// TIA Portal V19 export
FUNCTION_BLOCK "FeedMachine_FB"   // FB25, LAD
TITLE = FEEDING AXIS MACHINE
// stored: Access Published, MemoryReserve 100, SetENOAutomatically false
   VAR_INPUT
      AreaInterface : "AreaInterface";
      ZSI : "udt_ZoneSafetyInterface";
      DSI : "udt_DeviceSafetyInterface";
      Drive : "TAx_DriveInterface";
      DataIn : "FeedMachine_DataIn";
      CIn : "FeedMachine_CIn";
      Config : "FeedMachine_Config";
   END_VAR
   VAR_OUTPUT
      MachineInterface : "MachineInterface";
      DataOut : "FeedMachine_DataOut";
      COut : "FeedMachine_COut";
   END_VAR
   VAR_IN_OUT
      TO_Ax : TO_SpeedAxis;
      Par : "FeedMachine_Par";
      Alarm : "FeedMachine_Alr";
      Warning : "FeedMachine_Wng";
   END_VAR
   VAR
      Sts : Struct
         Standstill : Bool := TRUE;
         AlarmPresence : Bool := FALSE;
         WarningPresence : Bool := FALSE;
         Gen_Cnd : Bool;
         Bwd_Cnd : Bool := FALSE;
         Fwd_Cnd : Bool := FALSE;
         ReductionRatio : LReal := 1.0;
      END_STRUCT;
      Ctrl : Struct
         StopDueDoorOpeningRequest : Bool;
         StopInPhase : Bool;
         StopProgrammed : Bool;
         StopAborting : Bool;
         Man_HighSpeed : Bool;
         Bwd_Man : Bool;
         Fwd_Man : Bool;
         Bwd_Aut : Bool;
         Fwd_Aut : Bool;
         Fan : Bool;
         Vel : LReal;
         Acc : LReal;
         Dec : LReal;
         Jerk : LReal;
      END_STRUCT;
      Diag : Struct
         Ax : "TO_Diagnostic";
      END_STRUCT;
      Ax : "SpeedAxis";
      Fan_M : "Motor";
      TON_NoPendingCmd : TON_TIME;
      TON_Feed_DelayManChangeSpeed : TON_TIME;
      TON_MissingCndBwd { S7_SetPoint := 'True'} : TON_TIME;
      TON_MissingCndFwd { S7_SetPoint := 'True'} : TON_TIME;
      TON_Fan_DelayOff : TON_TIME;
      TON_Brake_TimeOut { S7_SetPoint := 'True'} : TON_TIME;
      AUX : Struct
         PB_Bwd : Bool;
         PB_Fwd : Bool;
      END_STRUCT;
   END_VAR
   VAR_TEMP
      PE : Struct
         PB_Bwd : Bool;
         PB_Fwd : Bool;
      END_STRUCT;
      Req : Bool;
      AxisVelMax : LReal;
      LimVel_EngUnit : LReal;
      LimAcc_EngUnit : LReal;
      LimDec_EngUnit : LReal;
      LimJerk_EngUnit : LReal;
      Real_VelTarget : LReal;
   END_VAR
   VAR_TEMP   // added for the SCL form of the ladder/FBD networks
      _w1 : Bool;
      _w2 : Bool;
   END_VAR
BEGIN

REGION Network 1 (SCL): Reset
   IF #AreaInterface.RstAlarms THEN

       #Alarm.BrakeTimeOut :=

       #Warning.NotAutReady :=
       #Warning.MissingCnd_Bkw :=
       #Warning.MissingCnd_Fwd := FALSE;
   END_IF;
END_REGION

REGION Network 2: Alarm motor brake timeout
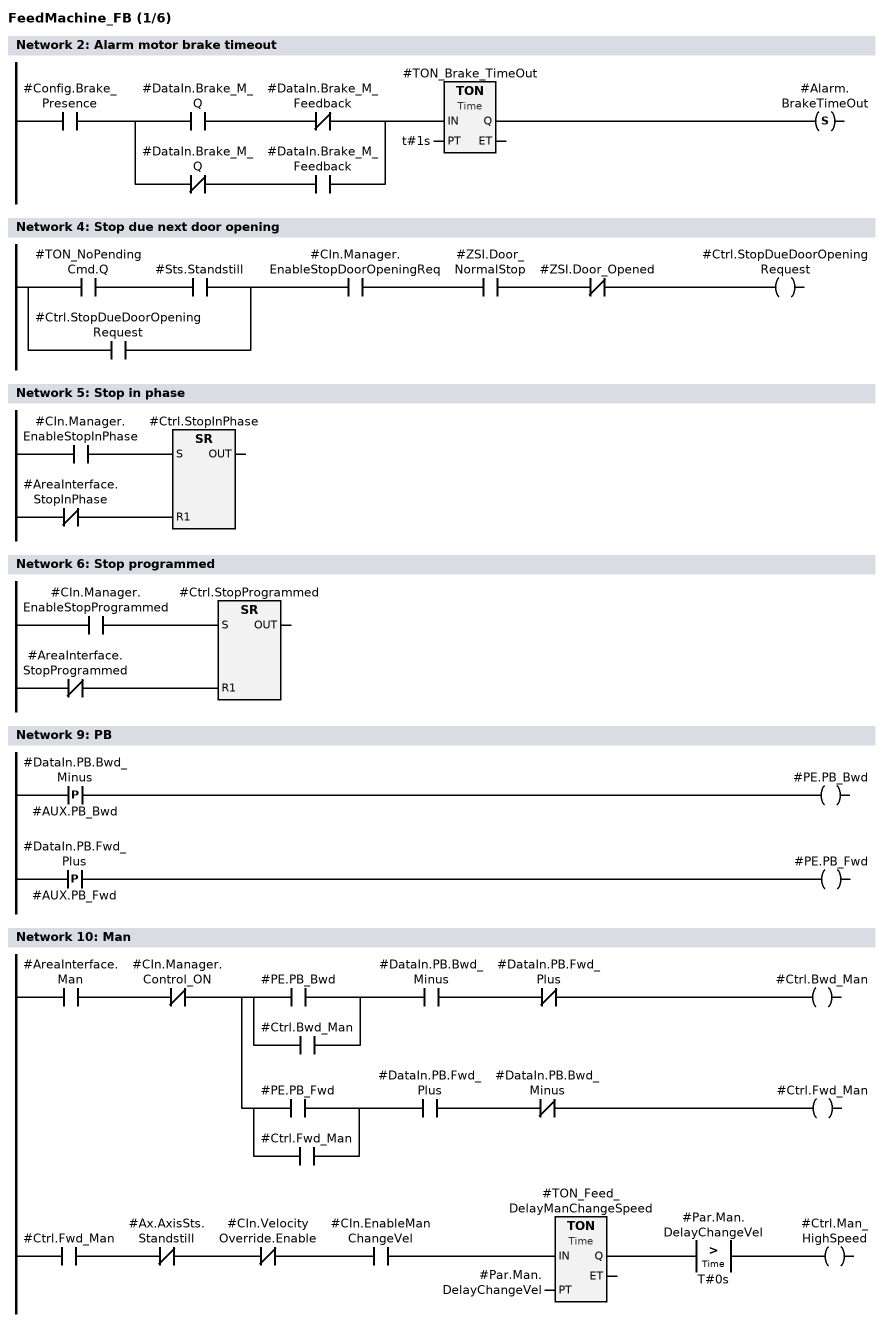
   RUNG wire#powerrail
      Contact( #Config.Brake_Presence )
      wire#w1
      Contact( #DataIn.Brake_M_Q )
      I_Contact( #DataIn.Brake_M_Feedback )
      wire#w2
      { S7_Templates := "time_type := Time" } #TON_Brake_TimeOut.TON(pt := t#1s, et =>)
      S_Coil( #Alarm.BrakeTimeOut )
   END_RUNG
   RUNG wire#w1
      I_Contact( #DataIn.Brake_M_Q )
      Contact( #DataIn.Brake_M_Feedback )
   END_RUNG wire#w2
   // the same network as SCL:
   #TON_Brake_TimeOut(IN := #Config.Brake_Presence AND ((#DataIn.Brake_M_Q AND NOT #DataIn.Brake_M_Feedback) OR (NOT #DataIn.Brake_M_Q AND #DataIn.Brake_M_Feedback)),   // TON
                      PT := t#1s);
   IF #TON_Brake_TimeOut.Q THEN #Alarm.BrakeTimeOut := TRUE; END_IF;
END_REGION

REGION Network 3: <<< MACHINE STOP >>>
END_REGION

REGION Network 4: Stop due next door opening
   RUNG wire#powerrail
      Contact( #TON_NoPendingCmd.Q )
      Contact( #Sts.Standstill )
      wire#w1
      Contact( #CIn.Manager.EnableStopDoorOpeningReq )
      Contact( #ZSI.Door_NormalStop )
      I_Contact( #ZSI.Door_Opened )
      Coil( #Ctrl.StopDueDoorOpeningRequest )
   END_RUNG
   RUNG wire#powerrail
      Contact( #Ctrl.StopDueDoorOpeningRequest )
   END_RUNG wire#w1
   // the same network as SCL:
   #Ctrl.StopDueDoorOpeningRequest := ((#TON_NoPendingCmd.Q AND #Sts.Standstill) OR #Ctrl.StopDueDoorOpeningRequest) AND #CIn.Manager.EnableStopDoorOpeningReq AND #ZSI.Door_NormalStop AND NOT #ZSI.Door_Opened;
END_REGION

REGION Network 5: Stop in phase
   RUNG wire#powerrail
      Contact( #CIn.Manager.EnableStopInPhase )
      S_SR(operand := #Ctrl.StopInPhase, r1 := wire#w1)
   END_RUNG
   RUNG wire#powerrail
      I_Contact( #AreaInterface.StopInPhase )
   END_RUNG wire#w1
   // the same network as SCL:
   IF #CIn.Manager.EnableStopInPhase THEN
       #Ctrl.StopInPhase := TRUE;   // SR flip-flop
   END_IF;
   IF NOT #AreaInterface.StopInPhase THEN #Ctrl.StopInPhase := FALSE; END_IF;
END_REGION

REGION Network 6: Stop programmed
   RUNG wire#powerrail
      Contact( #CIn.Manager.EnableStopProgrammed )
      S_SR(operand := #Ctrl.StopProgrammed, r1 := wire#w1)
   END_RUNG
   RUNG wire#powerrail
      I_Contact( #AreaInterface.StopProgrammed )
   END_RUNG wire#w1
   // the same network as SCL:
   IF #CIn.Manager.EnableStopProgrammed THEN
       #Ctrl.StopProgrammed := TRUE;   // SR flip-flop
   END_IF;
   IF NOT #AreaInterface.StopProgrammed THEN #Ctrl.StopProgrammed := FALSE; END_IF;
END_REGION

REGION Network 7: >
END_REGION

REGION Network 8: <<< FEED >>>
END_REGION

REGION Network 9: PB
   RUNG wire#powerrail
      P_Contact(operand := #DataIn.PB.Bwd_Minus, bit := #AUX.PB_Bwd)
      Coil( #PE.PB_Bwd )
   END_RUNG
   RUNG wire#powerrail
      P_Contact(operand := #DataIn.PB.Fwd_Plus, bit := #AUX.PB_Fwd)
      Coil( #PE.PB_Fwd )
   END_RUNG
   // the same network as SCL:
   #_w1 := #DataIn.PB.Bwd_Minus AND NOT #AUX.PB_Bwd;   // rising edge of #DataIn.PB.Bwd_Minus
   #AUX.PB_Bwd := #DataIn.PB.Bwd_Minus;
   #PE.PB_Bwd := #_w1;
   #_w2 := #DataIn.PB.Fwd_Plus AND NOT #AUX.PB_Fwd;   // rising edge of #DataIn.PB.Fwd_Plus
   #AUX.PB_Fwd := #DataIn.PB.Fwd_Plus;
   #PE.PB_Fwd := #_w2;
END_REGION

REGION Network 10: Man
   RUNG wire#powerrail
      Contact( #AreaInterface.Man )
      I_Contact( #CIn.Manager.Control_ON )
      wire#w1
      Contact( #PE.PB_Bwd )
      wire#w2
      Contact( #DataIn.PB.Bwd_Minus )
      I_Contact( #DataIn.PB.Fwd_Plus )
      Coil( #Ctrl.Bwd_Man )
   END_RUNG
   RUNG wire#w1
      Contact( #Ctrl.Bwd_Man )
   END_RUNG wire#w2
   RUNG wire#w1
      Contact( #PE.PB_Fwd )
      wire#w3
      Contact( #DataIn.PB.Fwd_Plus )
      I_Contact( #DataIn.PB.Bwd_Minus )
      Coil( #Ctrl.Fwd_Man )
   END_RUNG
   RUNG wire#w1
      Contact( #Ctrl.Fwd_Man )
   END_RUNG wire#w3
   RUNG wire#powerrail
      Contact( #Ctrl.Fwd_Man )
      I_Contact( #Ax.AxisSts.Standstill )
      I_Contact( #CIn.VelocityOverride.Enable )
      Contact( #CIn.EnableManChangeVel )
      { S7_Templates := "time_type := Time" } #TON_Feed_DelayManChangeSpeed.TON(pt := #Par.Man.DelayChangeVel, et =>)
      { S7_Templates := "SrcType := Time" } GT_Contact(in1 := #Par.Man.DelayChangeVel, in2 := T#0s)
      Coil( #Ctrl.Man_HighSpeed )
   END_RUNG
   // the same network as SCL:
   #_w1 := #AreaInterface.Man AND NOT #CIn.Manager.Control_ON;
   #Ctrl.Bwd_Man := #_w1 AND (#PE.PB_Bwd OR #Ctrl.Bwd_Man) AND #DataIn.PB.Bwd_Minus AND NOT #DataIn.PB.Fwd_Plus;
   #Ctrl.Fwd_Man := #_w1 AND (#PE.PB_Fwd OR #Ctrl.Fwd_Man) AND #DataIn.PB.Fwd_Plus AND NOT #DataIn.PB.Bwd_Minus;
   #TON_Feed_DelayManChangeSpeed(IN := #Ctrl.Fwd_Man AND NOT #Ax.AxisSts.Standstill AND NOT #CIn.VelocityOverride.Enable AND #CIn.EnableManChangeVel,   // TON
                           PT := #Par.Man.DelayChangeVel);
   #Ctrl.Man_HighSpeed := #TON_Feed_DelayManChangeSpeed.Q AND (#Par.Man.DelayChangeVel > T#0s);
END_REGION

REGION Network 11: Aut
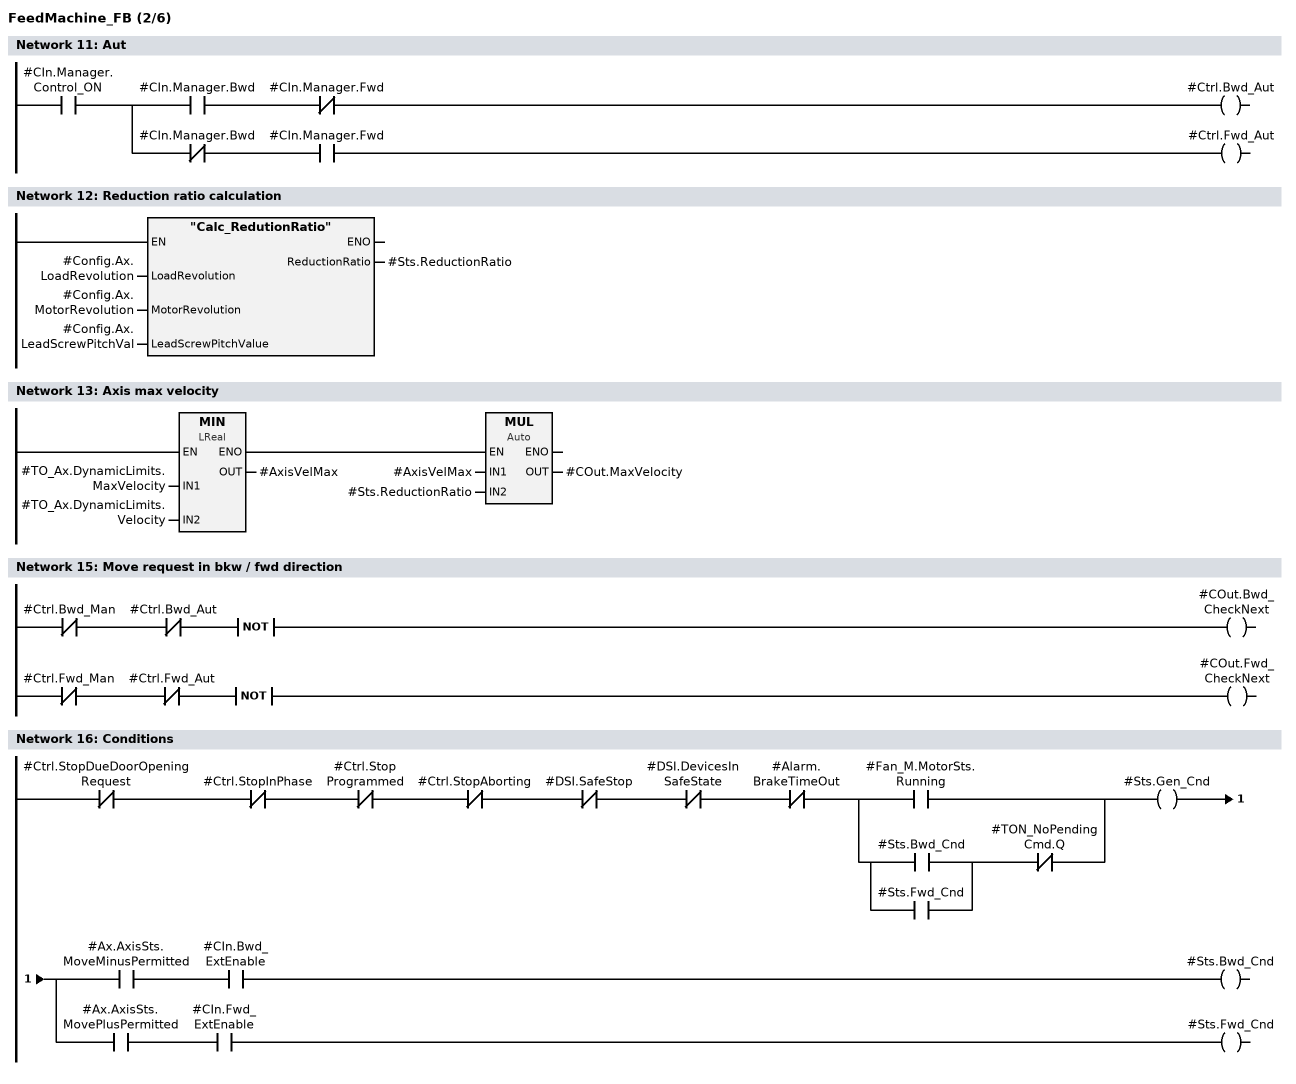
   RUNG wire#powerrail
      Contact( #CIn.Manager.Control_ON )
      wire#w1
      Contact( #CIn.Manager.Bwd )
      I_Contact( #CIn.Manager.Fwd )
      Coil( #Ctrl.Bwd_Aut )
   END_RUNG
   RUNG wire#w1
      I_Contact( #CIn.Manager.Bwd )
      Contact( #CIn.Manager.Fwd )
      Coil( #Ctrl.Fwd_Aut )
   END_RUNG
   // the same network as SCL:
   #Ctrl.Bwd_Aut := #CIn.Manager.Control_ON AND #CIn.Manager.Bwd AND NOT #CIn.Manager.Fwd;
   #Ctrl.Fwd_Aut := #CIn.Manager.Control_ON AND NOT #CIn.Manager.Bwd AND #CIn.Manager.Fwd;
END_REGION

REGION Network 12: Reduction ratio calculation
   RUNG wire#powerrail
      "Calc_RedutionRatio"(LoadRevolution := #Config.Ax.LoadRevolution, MotorRevolution := #Config.Ax.MotorRevolution, LeadScrewPitchValue := #Config.Ax.LeadScrewPitchVal, ReductionRatio => #Sts.ReductionRatio)
   END_RUNG
   // the same network as SCL:
   "Calc_RedutionRatio"(LoadRevolution := #Config.Ax.LoadRevolution,
                        MotorRevolution := #Config.Ax.MotorRevolution,
                        LeadScrewPitchValue := #Config.Ax.LeadScrewPitchVal,
                        ReductionRatio => #Sts.ReductionRatio);
END_REGION

REGION Network 13: Axis max velocity
   RUNG wire#powerrail
      { S7_Templates := "[card := 2, value_type := LReal]" } MIN(in1 := #TO_Ax.DynamicLimits.MaxVelocity, in2 := #TO_Ax.DynamicLimits.Velocity, out => #AxisVelMax)
      Mul(in1 := #AxisVelMax, in2 := #Sts.ReductionRatio, out => #COut.MaxVelocity)
   END_RUNG
   // the same network as SCL:
   #AxisVelMax := MIN(IN1 := #TO_Ax.DynamicLimits.MaxVelocity, IN2 := #TO_Ax.DynamicLimits.Velocity);
   #COut.MaxVelocity := #AxisVelMax * #Sts.ReductionRatio;
END_REGION

REGION Network 14 (SCL): Velocity & Dynamics
   #LimVel_EngUnit := #TO_Ax.DynamicLimits.MaxVelocity *  #Sts.ReductionRatio;
   #LimAcc_EngUnit := #TO_Ax.DynamicLimits.MaxAcceleration * #Sts.ReductionRatio;
   #LimDec_EngUnit := #TO_Ax.DynamicLimits.MaxDeceleration * #Sts.ReductionRatio;
   #LimJerk_EngUnit := #TO_Ax.DynamicLimits.MaxJerk * #Sts.ReductionRatio;




   #Ctrl.Vel := 0.0;

   IF #Ctrl.Bwd_Man AND #Ax.AxisCtrl.MoveMinus THEN


       #Ctrl.Acc := #Par.Man.Acc;
       #Ctrl.Dec := #Par.Man.Dec;
       #Ctrl.Jerk := #Par.Man.Jerk;

       #Ctrl.Vel := #Par.Man.VelBwd;

   ELSIF #Ctrl.Fwd_Man AND #Ax.AxisCtrl.MovePlus THEN


       #Ctrl.Acc := #Par.Man.Acc;
       #Ctrl.Dec := #Par.Man.Dec;
       #Ctrl.Jerk := #Par.Man.Jerk;


       IF #Ctrl.Man_HighSpeed THEN
           #Ctrl.Vel := #Par.Man.VelFwdHigh;
       ELSE
           #Ctrl.Vel := #Par.Man.VelFwdLow;
       END_IF;


   ELSIF (#Ctrl.Bwd_Aut AND #Ax.AxisCtrl.MoveMinus) OR (#Ctrl.Fwd_Aut AND #Ax.AxisCtrl.MovePlus)  THEN

       #Ctrl.Vel := #CIn.Manager.Vel;
       #Ctrl.Acc := #CIn.Manager.Acc;
       #Ctrl.Dec := #CIn.Manager.Dec;
       #Ctrl.Jerk := #CIn.Manager.Jerk;

   END_IF;


   // Dynamics limit

   #Ctrl.Vel := MIN(IN1:= #Ctrl.Vel,IN2:= #LimVel_EngUnit);

   #Ctrl.Acc := MIN(IN1:= #Ctrl.Acc,IN2:= #LimAcc_EngUnit);
   IF #Ctrl.Acc <= 0.0 THEN
       #Ctrl.Acc := #Par.Man.Acc;
   END_IF;

   #Ctrl.Dec := MIN(IN1:= #Ctrl.Dec,IN2:= #LimDec_EngUnit);
   IF #Ctrl.Dec <= 0.0 THEN
       #Ctrl.Dec := #Par.Man.Dec;
   END_IF;

   IF #Ctrl.Jerk > 0.0 THEN
       #Ctrl.Jerk := MIN(IN1:= #Ctrl.Jerk,IN2:= #LimJerk_EngUnit);
   ELSE
       #Ctrl.Jerk := 0.0;
   END_IF;



   // Velocity override
   // 
   #TO_Ax.Override.Velocity := 100.0;
   IF #CIn.VelocityOverride.Enable THEN
       #TO_Ax.Override.Velocity := LIMIT(MN:= 1.0, IN:=#CIn.VelocityOverride.Value, MX:=100.0);
   END_IF;



   // SLS velocity limit
   //
   IF #ZSI.Door_Opened AND #Ctrl.Vel > #Config.SLS_VEL THEN
       #Ctrl.Vel := #Config.SLS_VEL;
   END_IF;



   // Conversion and write dynamics value
   // 
   #Ax.AxisCtrl.Velocity := #Ctrl.Vel / #Sts.ReductionRatio;
   #Ax.AxisCtrl.Acceleration := #Ctrl.Acc / #Sts.ReductionRatio;
   #Ax.AxisCtrl.Deceleration := #Ctrl.Dec / #Sts.ReductionRatio;
   #Ax.AxisCtrl.Jerk := #Ctrl.Jerk / #Sts.ReductionRatio;

   #Ax.StandtillVelocity := #Config.Ax.StandstillVelocity / #Sts.ReductionRatio;
END_REGION

REGION Network 15: Move request in bkw / fwd direction
   RUNG wire#powerrail
      I_Contact( #Ctrl.Bwd_Man )
      I_Contact( #Ctrl.Bwd_Aut )
      Not()
      Coil( #COut.Bwd_CheckNext )
   END_RUNG
   RUNG wire#powerrail
      I_Contact( #Ctrl.Fwd_Man )
      I_Contact( #Ctrl.Fwd_Aut )
      Not()
      Coil( #COut.Fwd_CheckNext )
   END_RUNG
   // the same network as SCL:
   #COut.Bwd_CheckNext := NOT (NOT #Ctrl.Bwd_Man AND NOT #Ctrl.Bwd_Aut);
   #COut.Fwd_CheckNext := NOT (NOT #Ctrl.Fwd_Man AND NOT #Ctrl.Fwd_Aut);
END_REGION

REGION Network 16: Conditions
   RUNG wire#powerrail
      I_Contact( #Ctrl.StopDueDoorOpeningRequest )
      I_Contact( #Ctrl.StopInPhase )
      I_Contact( #Ctrl.StopProgrammed )
      I_Contact( #Ctrl.StopAborting )
      I_Contact( #DSI.SafeStop )
      I_Contact( #DSI.DevicesInSafeState )
      I_Contact( #Alarm.BrakeTimeOut )
      wire#w1
      Contact( #Fan_M.MotorSts.Running )
      wire#w2
      Coil( #Sts.Gen_Cnd )
      wire#w4
      Contact( #Ax.AxisSts.MoveMinusPermitted )
      Contact( #CIn.Bwd_ExtEnable )
      Coil( #Sts.Bwd_Cnd )
   END_RUNG
   RUNG wire#w1
      Contact( #Sts.Bwd_Cnd )
      wire#w3
      I_Contact( #TON_NoPendingCmd.Q )
   END_RUNG wire#w2
   RUNG wire#w1
      Contact( #Sts.Fwd_Cnd )
   END_RUNG wire#w3
   RUNG wire#w4
      Contact( #Ax.AxisSts.MovePlusPermitted )
      Contact( #CIn.Fwd_ExtEnable )
      Coil( #Sts.Fwd_Cnd )
   END_RUNG
   // the same network as SCL:
   #Sts.Gen_Cnd := NOT #Ctrl.StopDueDoorOpeningRequest AND NOT #Ctrl.StopInPhase AND NOT #Ctrl.StopProgrammed AND NOT #Ctrl.StopAborting AND NOT #DSI.SafeStop AND NOT #DSI.DevicesInSafeState AND NOT #Alarm.BrakeTimeOut AND (#Fan_M.MotorSts.Running OR ((#Sts.Bwd_Cnd OR #Sts.Fwd_Cnd) AND NOT #TON_NoPendingCmd.Q));
   #Sts.Bwd_Cnd := #Sts.Gen_Cnd AND #Ax.AxisSts.MoveMinusPermitted AND #CIn.Bwd_ExtEnable;
   #Sts.Fwd_Cnd := #Sts.Gen_Cnd AND #Ax.AxisSts.MovePlusPermitted AND #CIn.Fwd_ExtEnable;
END_REGION

REGION Network 17: Missing conditions
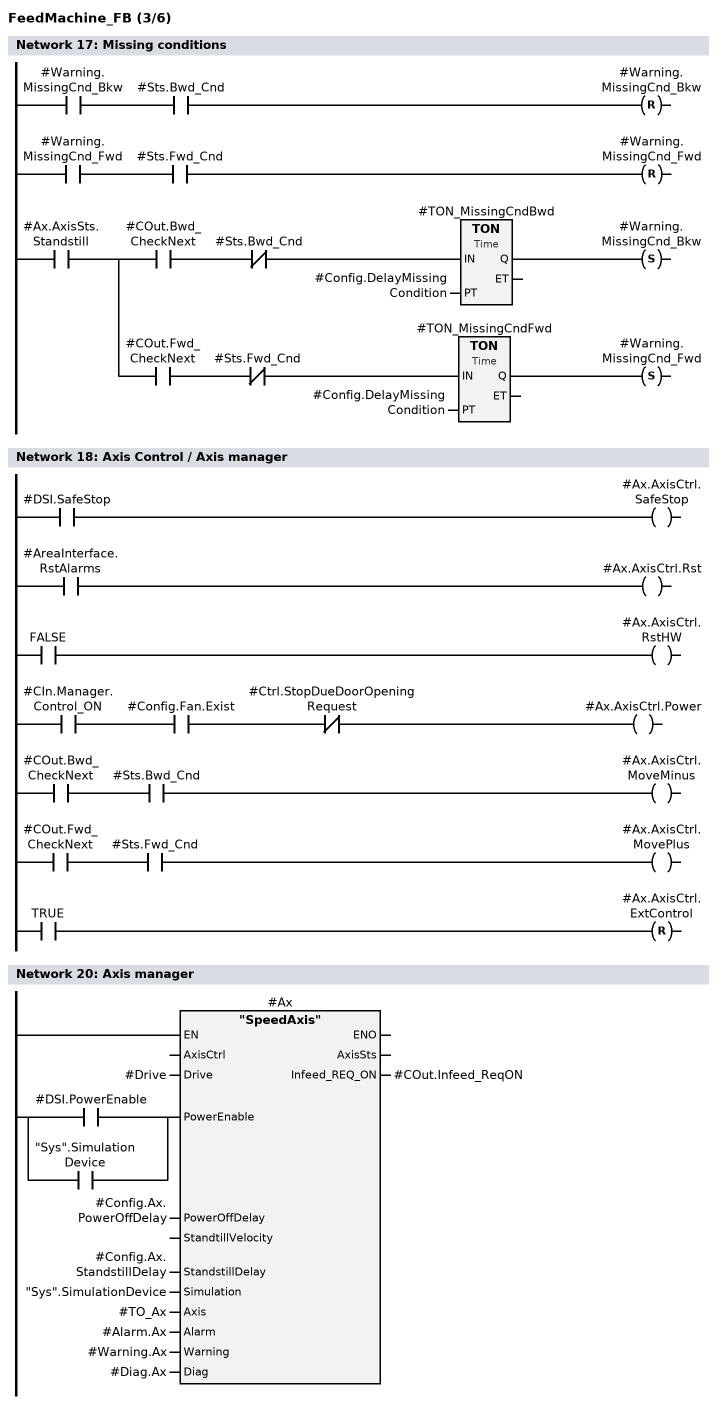
   RUNG wire#powerrail
      Contact( #Warning.MissingCnd_Bkw )
      Contact( #Sts.Bwd_Cnd )
      R_Coil( #Warning.MissingCnd_Bkw )
   END_RUNG
   RUNG wire#powerrail
      Contact( #Warning.MissingCnd_Fwd )
      Contact( #Sts.Fwd_Cnd )
      R_Coil( #Warning.MissingCnd_Fwd )
   END_RUNG
   RUNG wire#powerrail
      Contact( #Ax.AxisSts.Standstill )
      wire#w1
      Contact( #COut.Bwd_CheckNext )
      I_Contact( #Sts.Bwd_Cnd )
      { S7_Templates := "time_type := Time" } #TON_MissingCndBwd.TON(pt := #Config.DelayMissingCondition, et =>)
      S_Coil( #Warning.MissingCnd_Bkw )
   END_RUNG
   RUNG wire#w1
      Contact( #COut.Fwd_CheckNext )
      I_Contact( #Sts.Fwd_Cnd )
      { S7_Templates := "time_type := Time" } #TON_MissingCndFwd.TON(pt := #Config.DelayMissingCondition, et =>)
      S_Coil( #Warning.MissingCnd_Fwd )
   END_RUNG
   // the same network as SCL:
   IF #Warning.MissingCnd_Bkw AND #Sts.Bwd_Cnd THEN #Warning.MissingCnd_Bkw := FALSE; END_IF;
   IF #Warning.MissingCnd_Fwd AND #Sts.Fwd_Cnd THEN #Warning.MissingCnd_Fwd := FALSE; END_IF;
   #TON_MissingCndBwd(IN := #Ax.AxisSts.Standstill AND #COut.Bwd_CheckNext AND NOT #Sts.Bwd_Cnd,   // TON
                      PT := #Config.DelayMissingCondition);
   IF #TON_MissingCndBwd.Q THEN #Warning.MissingCnd_Bkw := TRUE; END_IF;
   #TON_MissingCndFwd(IN := #Ax.AxisSts.Standstill AND #COut.Fwd_CheckNext AND NOT #Sts.Fwd_Cnd,   // TON
                      PT := #Config.DelayMissingCondition);
   IF #TON_MissingCndFwd.Q THEN #Warning.MissingCnd_Fwd := TRUE; END_IF;
END_REGION

REGION Network 18: Axis Control / Axis manager
   RUNG wire#powerrail
      Contact( #DSI.SafeStop )
      Coil( #Ax.AxisCtrl.SafeStop )
   END_RUNG
   RUNG wire#powerrail
      Contact( #AreaInterface.RstAlarms )
      Coil( #Ax.AxisCtrl.Rst )
   END_RUNG
   RUNG wire#powerrail
      Contact( FALSE )
      Coil( #Ax.AxisCtrl.RstHW )
   END_RUNG
   RUNG wire#powerrail
      Contact( #CIn.Manager.Control_ON )
      Contact( #Config.Fan.Exist )
      I_Contact( #Ctrl.StopDueDoorOpeningRequest )
      Coil( #Ax.AxisCtrl.Power )
   END_RUNG
   RUNG wire#powerrail
      Contact( #COut.Bwd_CheckNext )
      Contact( #Sts.Bwd_Cnd )
      Coil( #Ax.AxisCtrl.MoveMinus )
   END_RUNG
   RUNG wire#powerrail
      Contact( #COut.Fwd_CheckNext )
      Contact( #Sts.Fwd_Cnd )
      Coil( #Ax.AxisCtrl.MovePlus )
   END_RUNG
   RUNG wire#powerrail
      Contact( TRUE )
      R_Coil( #Ax.AxisCtrl.ExtControl )
   END_RUNG
   // the same network as SCL:
   #Ax.AxisCtrl.SafeStop := #DSI.SafeStop;
   #Ax.AxisCtrl.Rst := #AreaInterface.RstAlarms;
   #Ax.AxisCtrl.RstHW := FALSE;
   #Ax.AxisCtrl.Power := #CIn.Manager.Control_ON AND #Config.Fan.Exist AND NOT #Ctrl.StopDueDoorOpeningRequest;
   #Ax.AxisCtrl.MoveMinus := #COut.Bwd_CheckNext AND #Sts.Bwd_Cnd;
   #Ax.AxisCtrl.MovePlus := #COut.Fwd_CheckNext AND #Sts.Fwd_Cnd;
   IF TRUE THEN #Ax.AxisCtrl.ExtControl := FALSE; END_IF;
END_REGION

REGION Network 20: Axis manager
   RUNG wire#powerrail
      #Ax(PowerEnable := wire#w1, AxisCtrl :=, Drive := #Drive, PowerOffDelay := #Config.Ax.PowerOffDelay, StandtillVelocity :=, StandstillDelay := #Config.Ax.StandstillDelay, Simulation := "Sys".SimulationDevice, Axis := #TO_Ax, Alarm := #Alarm.Ax, Warning := #Warning.Ax, Diag := #Diag.Ax, AxisSts =>, Infeed_REQ_ON => #COut.Infeed_ReqON)
   END_RUNG
   RUNG wire#powerrail
      Contact( #DSI.PowerEnable )
   END_RUNG wire#w1
   RUNG wire#powerrail
      Contact( "Sys".SimulationDevice )
   END_RUNG wire#w1
   // the same network as SCL:
   #Ax(Drive := #Drive,   // "SpeedAxis"
       PowerEnable := #DSI.PowerEnable OR "Sys".SimulationDevice,
       PowerOffDelay := #Config.Ax.PowerOffDelay,
       StandstillDelay := #Config.Ax.StandstillDelay,
       Simulation := "Sys".SimulationDevice,
       Axis := #TO_Ax,
       Alarm := #Alarm.Ax,
       Warning := #Warning.Ax,
       Diag := #Diag.Ax,
       Infeed_REQ_ON => #COut.Infeed_ReqON);
END_REGION

REGION Network 21: Mask warning 1699 = Test stop STO required
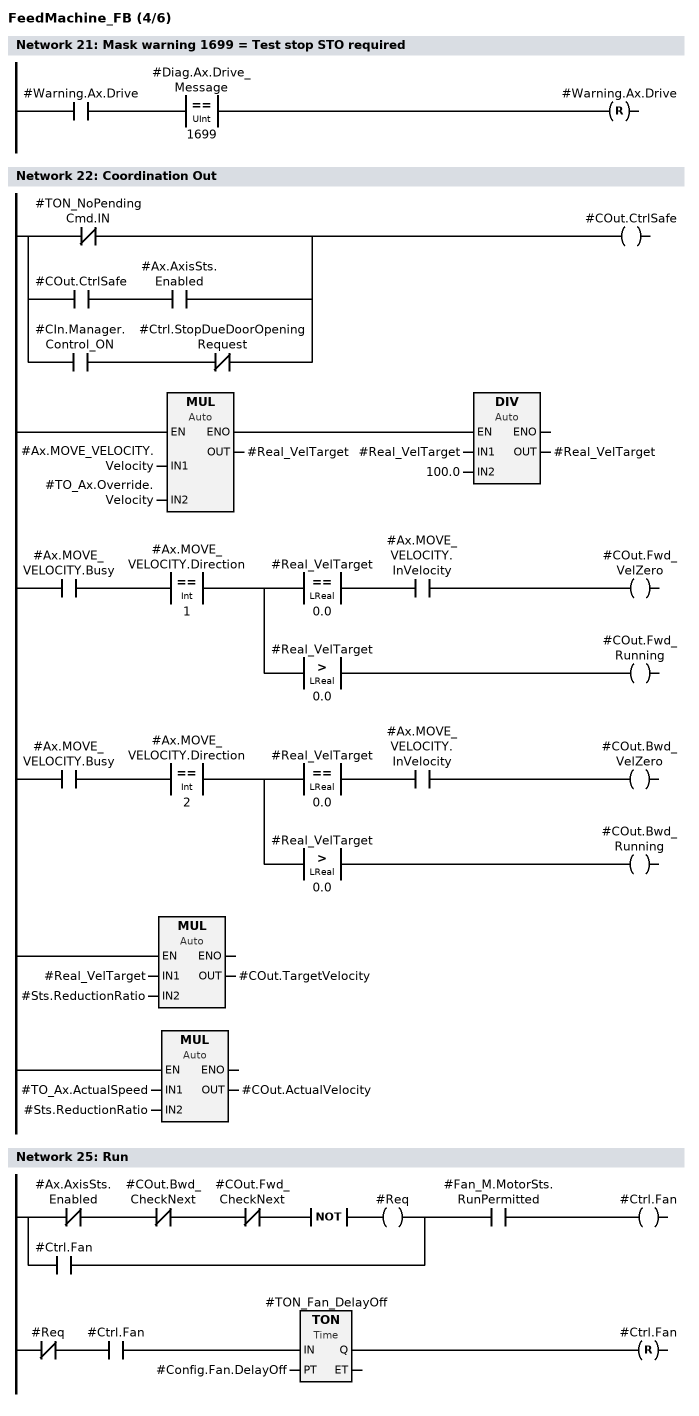
   RUNG wire#powerrail
      Contact( #Warning.Ax.Drive )
      { S7_Templates := "SrcType := UInt" } EQ_Contact(in1 := #Diag.Ax.Drive_Message, in2 := 1699)
      R_Coil( #Warning.Ax.Drive )
   END_RUNG
   // the same network as SCL:
   IF #Warning.Ax.Drive AND (#Diag.Ax.Drive_Message = 1699) THEN #Warning.Ax.Drive := FALSE; END_IF;
END_REGION

REGION Network 22: Coordination Out
   RUNG wire#powerrail
      I_Contact( #TON_NoPendingCmd.IN )
      wire#w1
      Coil( #COut.CtrlSafe )
   END_RUNG
   RUNG wire#powerrail
      Contact( #COut.CtrlSafe )
      Contact( #Ax.AxisSts.Enabled )
   END_RUNG wire#w1
   RUNG wire#powerrail
      Contact( #CIn.Manager.Control_ON )
      I_Contact( #Ctrl.StopDueDoorOpeningRequest )
   END_RUNG wire#w1
   RUNG wire#powerrail
      { S7_GenerateENO := "TRUE" } Mul(in1 := #Ax.MOVE_VELOCITY.Velocity, in2 := #TO_Ax.Override.Velocity, out => #Real_VelTarget)
      { S7_GenerateENO := "TRUE" } Div(in1 := #Real_VelTarget, in2 := 100.0, out => #Real_VelTarget)
   END_RUNG
   RUNG wire#powerrail
      Contact( #Ax.MOVE_VELOCITY.Busy )
      { S7_Templates := "SrcType := Int" } EQ_Contact(in1 := #Ax.MOVE_VELOCITY.Direction, in2 := 1)
      wire#w2
      { S7_Templates := "SrcType := LReal" } EQ_Contact(in1 := #Real_VelTarget, in2 := 0.0)
      Contact( #Ax.MOVE_VELOCITY.InVelocity )
      Coil( #COut.Fwd_VelZero )
   END_RUNG
   RUNG wire#w2
      { S7_Templates := "SrcType := LReal" } GT_Contact(in1 := #Real_VelTarget, in2 := 0.0)
      Coil( #COut.Fwd_Running )
   END_RUNG
   RUNG wire#powerrail
      Contact( #Ax.MOVE_VELOCITY.Busy )
      { S7_Templates := "SrcType := Int" } EQ_Contact(in1 := #Ax.MOVE_VELOCITY.Direction, in2 := 2)
      wire#w3
      { S7_Templates := "SrcType := LReal" } EQ_Contact(in1 := #Real_VelTarget, in2 := 0.0)
      Contact( #Ax.MOVE_VELOCITY.InVelocity )
      Coil( #COut.Bwd_VelZero )
   END_RUNG
   RUNG wire#w3
      { S7_Templates := "SrcType := LReal" } GT_Contact(in1 := #Real_VelTarget, in2 := 0.0)
      Coil( #COut.Bwd_Running )
   END_RUNG
   RUNG wire#powerrail
      { S7_GenerateENO := "TRUE" } Mul(in1 := #Real_VelTarget, in2 := #Sts.ReductionRatio, out => #COut.TargetVelocity)
   END_RUNG
   RUNG wire#powerrail
      { S7_GenerateENO := "TRUE" } Mul(in1 := #TO_Ax.ActualSpeed, in2 := #Sts.ReductionRatio, out => #COut.ActualVelocity)
   END_RUNG
   // the same network as SCL:
   // ENO of a box is taken as its EN; it also drops when the box reports an error
   #COut.CtrlSafe := NOT #TON_NoPendingCmd.IN OR (#COut.CtrlSafe AND #Ax.AxisSts.Enabled) OR (#CIn.Manager.Control_ON AND NOT #Ctrl.StopDueDoorOpeningRequest);
   #Real_VelTarget := #Ax.MOVE_VELOCITY.Velocity * #TO_Ax.Override.Velocity;
   #Real_VelTarget := #Real_VelTarget / 100.0;
   #_w1 := #Ax.MOVE_VELOCITY.Busy AND (#Ax.MOVE_VELOCITY.Direction = 1);
   #COut.Fwd_VelZero := #_w1 AND (#Real_VelTarget = 0.0) AND #Ax.MOVE_VELOCITY.InVelocity;
   #COut.Fwd_Running := #_w1 AND (#Real_VelTarget > 0.0);
   #_w2 := #Ax.MOVE_VELOCITY.Busy AND (#Ax.MOVE_VELOCITY.Direction = 2);
   #COut.Bwd_VelZero := #_w2 AND (#Real_VelTarget = 0.0) AND #Ax.MOVE_VELOCITY.InVelocity;
   #COut.Bwd_Running := #_w2 AND (#Real_VelTarget > 0.0);
   #COut.TargetVelocity := #Real_VelTarget * #Sts.ReductionRatio;
   #COut.ActualVelocity := #TO_Ax.ActualSpeed * #Sts.ReductionRatio;
END_REGION

REGION Network 23: >
END_REGION

REGION Network 24: <<< MOTOR FAN >>>
END_REGION

REGION Network 25: Run
   RUNG wire#powerrail
      I_Contact( #Ax.AxisSts.Enabled )
      I_Contact( #COut.Bwd_CheckNext )
      I_Contact( #COut.Fwd_CheckNext )
      Not()
      Coil( #Req )
      wire#w1
      Contact( #Fan_M.MotorSts.RunPermitted )
      Coil( #Ctrl.Fan )
   END_RUNG
   RUNG wire#powerrail
      Contact( #Ctrl.Fan )
   END_RUNG wire#w1
   RUNG wire#powerrail
      I_Contact( #Req )
      Contact( #Ctrl.Fan )
      { S7_Templates := "time_type := Time" } #TON_Fan_DelayOff.TON(pt := #Config.Fan.DelayOff, et =>)
      R_Coil( #Ctrl.Fan )
   END_RUNG
   // the same network as SCL:
   #Req := NOT (NOT #Ax.AxisSts.Enabled AND NOT #COut.Bwd_CheckNext AND NOT #COut.Fwd_CheckNext);
   #Ctrl.Fan := (#Req OR #Ctrl.Fan) AND #Fan_M.MotorSts.RunPermitted;
   #TON_Fan_DelayOff(IN := NOT #Req AND #Ctrl.Fan, PT := #Config.Fan.DelayOff);   // TON
   IF #TON_Fan_DelayOff.Q THEN #Ctrl.Fan := FALSE; END_IF;
END_REGION

REGION Network 26: Device
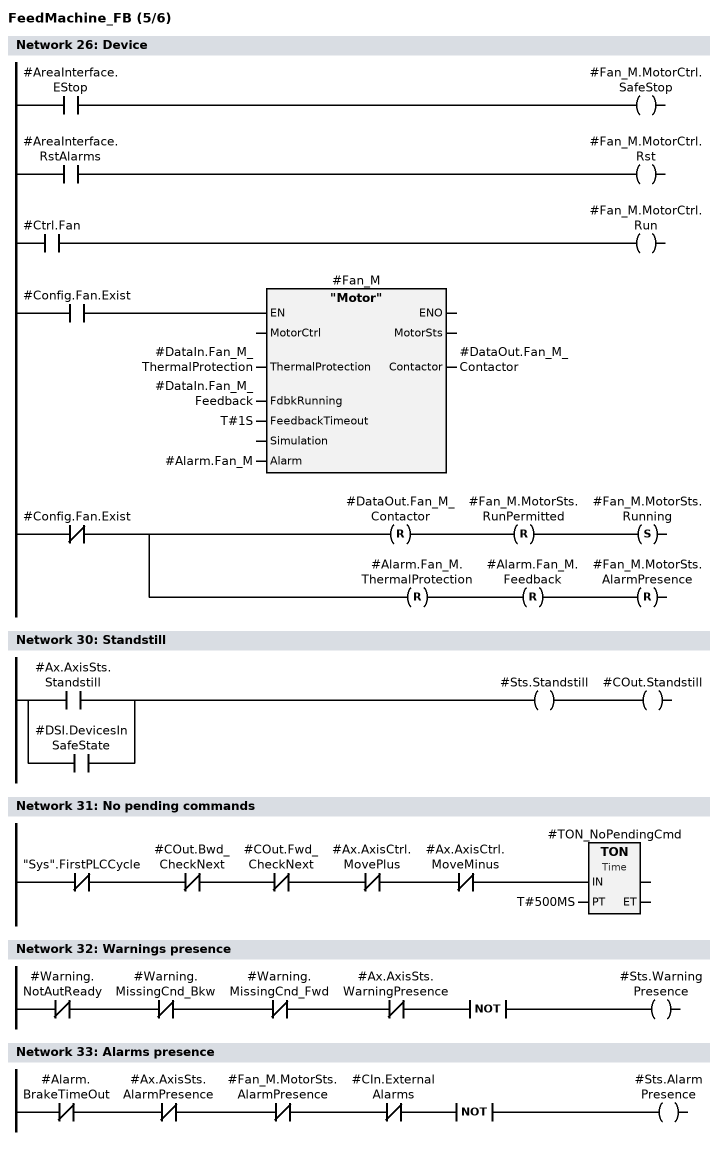
   RUNG wire#powerrail
      Contact( #AreaInterface.EStop )
      Coil( #Fan_M.MotorCtrl.SafeStop )
   END_RUNG
   RUNG wire#powerrail
      Contact( #AreaInterface.RstAlarms )
      Coil( #Fan_M.MotorCtrl.Rst )
   END_RUNG
   RUNG wire#powerrail
      Contact( #Ctrl.Fan )
      Coil( #Fan_M.MotorCtrl.Run )
   END_RUNG
   RUNG wire#powerrail
      Contact( #Config.Fan.Exist )
      #Fan_M(MotorCtrl :=, ThermalProtection := #DataIn.Fan_M_ThermalProtection, FdbkRunning := #DataIn.Fan_M_Feedback, FeedbackTimeout := T#1S, Simulation :=, Alarm := #Alarm.Fan_M, MotorSts =>, Contactor => #DataOut.Fan_M_Contactor)
   END_RUNG
   RUNG wire#powerrail
      I_Contact( #Config.Fan.Exist )
      wire#w1
      R_Coil( #DataOut.Fan_M_Contactor )
      R_Coil( #Fan_M.MotorSts.RunPermitted )
      S_Coil( #Fan_M.MotorSts.Running )
   END_RUNG
   RUNG wire#w1
      R_Coil( #Alarm.Fan_M.ThermalProtection )
      R_Coil( #Alarm.Fan_M.Feedback )
      R_Coil( #Fan_M.MotorSts.AlarmPresence )
   END_RUNG
   // the same network as SCL:
   #Fan_M.MotorCtrl.SafeStop := #AreaInterface.EStop;
   #Fan_M.MotorCtrl.Rst := #AreaInterface.RstAlarms;
   #Fan_M.MotorCtrl.Run := #Ctrl.Fan;
   IF #Config.Fan.Exist THEN
       #Fan_M(ThermalProtection := #DataIn.Fan_M_ThermalProtection,   // "Motor"
              FdbkRunning := #DataIn.Fan_M_Feedback,
              FeedbackTimeout := T#1S,
              Alarm := #Alarm.Fan_M,
              Contactor => #DataOut.Fan_M_Contactor);
   END_IF;
   IF NOT #Config.Fan.Exist THEN
       #DataOut.Fan_M_Contactor := FALSE;
       #Fan_M.MotorSts.RunPermitted := FALSE;
       #Fan_M.MotorSts.Running := TRUE;
       #Alarm.Fan_M.ThermalProtection := FALSE;
       #Alarm.Fan_M.Feedback := FALSE;
       #Fan_M.MotorSts.AlarmPresence := FALSE;
   END_IF;
END_REGION

REGION Network 27: >
END_REGION

REGION Network 28: >
END_REGION

REGION Network 29: <<< MACHINE STATUS >>>
END_REGION

REGION Network 30: Standstill
   RUNG wire#powerrail
      Contact( #Ax.AxisSts.Standstill )
      wire#w1
      Coil( #Sts.Standstill )
      Coil( #COut.Standstill )
   END_RUNG
   RUNG wire#powerrail
      Contact( #DSI.DevicesInSafeState )
   END_RUNG wire#w1
   // the same network as SCL:
   #Sts.Standstill := #Ax.AxisSts.Standstill OR #DSI.DevicesInSafeState;
   #COut.Standstill := #Sts.Standstill;
END_REGION

REGION Network 31: No pending commands
   RUNG wire#powerrail
      I_Contact( "Sys".FirstPLCCycle )
      I_Contact( #COut.Bwd_CheckNext )
      I_Contact( #COut.Fwd_CheckNext )
      I_Contact( #Ax.AxisCtrl.MovePlus )
      I_Contact( #Ax.AxisCtrl.MoveMinus )
      { S7_Templates := "time_type := Time" } #TON_NoPendingCmd.TON(pt := T#500MS, et =>)
   END_RUNG
   // the same network as SCL:
   #TON_NoPendingCmd(IN := NOT "Sys".FirstPLCCycle AND NOT #COut.Bwd_CheckNext AND NOT #COut.Fwd_CheckNext AND NOT #Ax.AxisCtrl.MovePlus AND NOT #Ax.AxisCtrl.MoveMinus,   // TON
                     PT := T#500MS);
END_REGION

REGION Network 32: Warnings presence
   RUNG wire#powerrail
      I_Contact( #Warning.NotAutReady )
      I_Contact( #Warning.MissingCnd_Bkw )
      I_Contact( #Warning.MissingCnd_Fwd )
      I_Contact( #Ax.AxisSts.WarningPresence )
      Not()
      Coil( #Sts.WarningPresence )
   END_RUNG
   // the same network as SCL:
   #Sts.WarningPresence := NOT (NOT #Warning.NotAutReady AND NOT #Warning.MissingCnd_Bkw AND NOT #Warning.MissingCnd_Fwd AND NOT #Ax.AxisSts.WarningPresence);
END_REGION

REGION Network 33: Alarms presence
   RUNG wire#powerrail
      I_Contact( #Alarm.BrakeTimeOut )
      I_Contact( #Ax.AxisSts.AlarmPresence )
      I_Contact( #Fan_M.MotorSts.AlarmPresence )
      I_Contact( #CIn.ExternalAlarms )
      Not()
      Coil( #Sts.AlarmPresence )
   END_RUNG
   // the same network as SCL:
   #Sts.AlarmPresence := NOT (NOT #Alarm.BrakeTimeOut AND NOT #Ax.AxisSts.AlarmPresence AND NOT #Fan_M.MotorSts.AlarmPresence AND NOT #CIn.ExternalAlarms);
END_REGION

REGION Network 34: Stop aborting
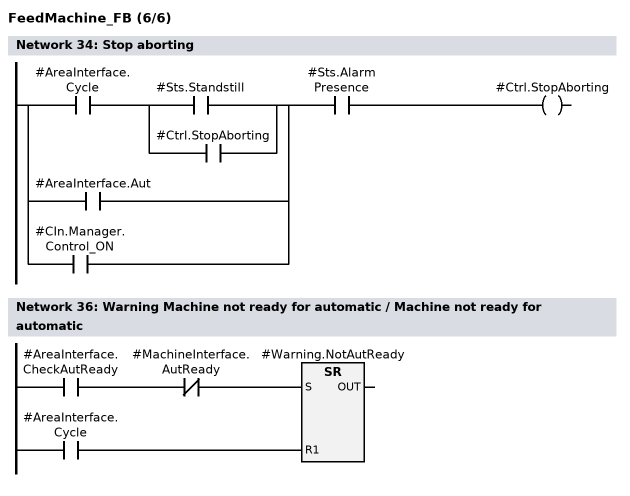
   RUNG wire#powerrail
      Contact( #AreaInterface.Cycle )
      wire#w1
      Contact( #Sts.Standstill )
      wire#w2
      Contact( #Sts.AlarmPresence )
      Coil( #Ctrl.StopAborting )
   END_RUNG
   RUNG wire#w1
      Contact( #Ctrl.StopAborting )
   END_RUNG wire#w2
   RUNG wire#powerrail
      Contact( #AreaInterface.Aut )
   END_RUNG wire#w2
   RUNG wire#powerrail
      Contact( #CIn.Manager.Control_ON )
   END_RUNG wire#w2
   // the same network as SCL:
   #Ctrl.StopAborting := ((#AreaInterface.Cycle AND (#Sts.Standstill OR #Ctrl.StopAborting)) OR #AreaInterface.Aut OR #CIn.Manager.Control_ON) AND #Sts.AlarmPresence;
END_REGION

REGION Network 35 (SCL): Collect machine to zone interface
   #MachineInterface.AutReady := #AreaInterface.Aut AND NOT #Sts.AlarmPresence;
   #MachineInterface.Aborting := #Ctrl.StopAborting;
   #MachineInterface.MotionsStandStill := #TON_NoPendingCmd.Q AND #Sts.Standstill;
   #MachineInterface.AckStopInPhase := #Ctrl.StopInPhase AND #MachineInterface.MotionsStandStill;
   #MachineInterface.AckStopProgrammed := #Ctrl.StopProgrammed AND #MachineInterface.MotionsStandStill;
   #MachineInterface.AlarmsPresence := #Sts.AlarmPresence;
   #MachineInterface.WarningPresence := #Sts.WarningPresence;
END_REGION

REGION Network 36: Warning Machine not ready for automatic / Machine not ready for automatic
   RUNG wire#powerrail
      Contact( #AreaInterface.CheckAutReady )
      I_Contact( #MachineInterface.AutReady )
      S_SR(operand := #Warning.NotAutReady, r1 := wire#w1)
   END_RUNG
   RUNG wire#powerrail
      Contact( #AreaInterface.Cycle )
   END_RUNG wire#w1
   // the same network as SCL:
   IF #AreaInterface.CheckAutReady AND NOT #MachineInterface.AutReady THEN
       #Warning.NotAutReady := TRUE;   // SR flip-flop
   END_IF;
   IF #AreaInterface.Cycle THEN #Warning.NotAutReady := FALSE; END_IF;
END_REGION

REGION Network 37: >
END_REGION

REGION Network 38: >
END_REGION

REGION Network 39: >
END_REGION
END_FUNCTION_BLOCK
